// LS Electric XG5000 project: 16-46-2
// PLC NewPLC
// module base 0 slot 0: 입출력 모듈:XBC-DR14E (DC 24V 입력 8점, 릴레이 출력 6점)

PROGRAM NewProgram (task: 스캔 프로그램)

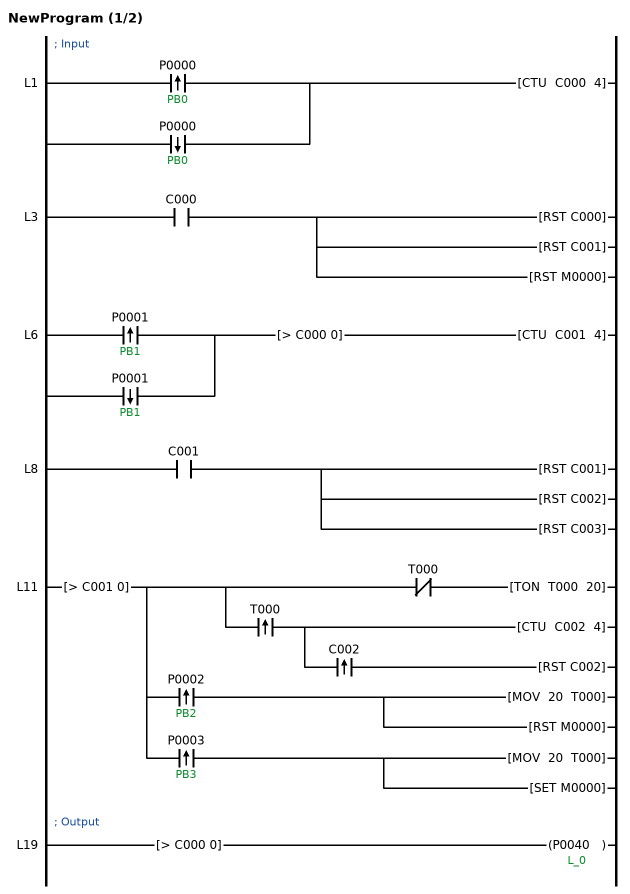
// Input
; L1
LOADP     P0000	// PB0
ORN       P0000	// PB0
CTU       C000 4
; L3
LOAD      C000
RST       C000
RST       C001
RST       M0000
; L6
LOADP     P0001	// PB1
ORN       P0001	// PB1
AND>      C000 0
CTU       C001 4
; L8
LOAD      C001
RST       C001
RST       C002
RST       C003
; L11
LOAD>     C001 0
MPUSH
AND NOT   T000
TON       T000 20
MLOAD
ANDP      T000
CTU       C002 4
ANDP      C002
RST       C002
MLOAD
ANDP      P0002	// PB2
MOV       20 T000
RST       M0000
MPOP
ANDP      P0003	// PB3
MOV       20 T000
SET       M0000
// Output
; L19
LOAD>     C000 0
OUT       P0040	// L_0

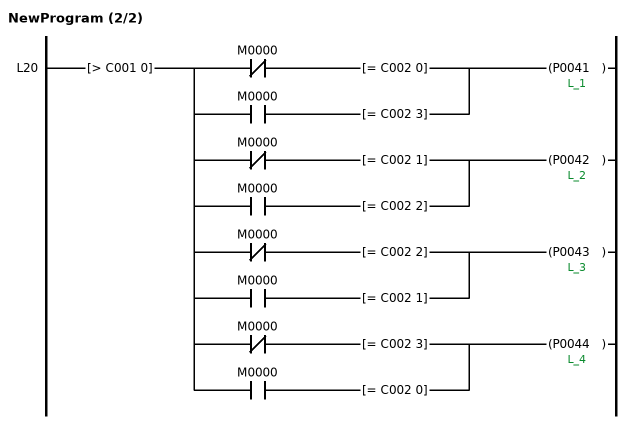
; L20
LOAD>     C001 0
MPUSH
LOAD NOT  M0000
AND=      C002 0
LOAD      M0000
AND=      C002 3
OR LOAD
AND LOAD
OUT       P0041	// L_1
MLOAD
LOAD NOT  M0000
AND=      C002 1
LOAD      M0000
AND=      C002 2
OR LOAD
AND LOAD
OUT       P0042	// L_2
MLOAD
LOAD NOT  M0000
AND=      C002 2
LOAD      M0000
AND=      C002 1
OR LOAD
AND LOAD
OUT       P0043	// L_3
MPOP
LOAD NOT  M0000
AND=      C002 3
LOAD      M0000
AND=      C002 0
OR LOAD
AND LOAD
OUT       P0044	// L_4